// TIA Portal V18 export
VAR_GLOBAL   // PLC tag table "Default tag table_1"
   System_Byte AT %MB1 : Byte;
   FirstScan AT %M1.0 : Bool;
   DiagStatusUpdate AT %M1.1 : Bool;
   AlwaysTRUE AT %M1.2 : Bool;
   AlwaysFALSE AT %M1.3 : Bool;
   Clock_Byte AT %MB0 : Byte;
   Clock_10Hz AT %M0.0 : Bool;
   Clock_5Hz AT %M0.1 : Bool;
   "Clock_2.5Hz" AT %M0.2 : Bool;
   Clock_2Hz AT %M0.3 : Bool;
   "Clock_1.25Hz" AT %M0.4 : Bool;
   Clock_1Hz AT %M0.5 : Bool;
   "Clock_0.625Hz" AT %M0.6 : Bool;
   "Clock_0.5Hz" AT %M0.7 : Bool;
   "H/SSR_019_START" AT %M2.0 : Bool;
   "H/SSR_019_SP" AT %MD4 : Real;
   "H/SSR_019_TT01_PV" AT %MD8 : Real;
   "H/SSR_019_ALERT_SP" AT %MD12 : Real;
   "H/SSR_019_CHBr_RT_SP" AT %MD16 : Real;
   "H/SSR_019_RT_HW_SP" AT %MD20 : Real;
   "H/SSR_019_HW_STEAM_SP" AT %MD24 : Real;
   "H/SSR_019_RT_CHBr_SP" AT %MD28 : Real;
   "H/SSR_019_SOURCE_SEL" AT %MW32 : Int;
   "H/SSR_019_AM" AT %M2.1 : Bool;
   "H/SSR_019_TIME_SP" AT %MW34 : Int;
   "H/SSR_019_KP" AT %MW36 : Int;
   "H/SSR_019_TI" AT %MW38 : Int;
   "H/SSR_019_TT02_PV" AT %MD40 : Real;
   "H/SSR_019_CV02_MANOUT" AT %MD44 : Real;
   "H/SSR_019_START_PV" AT %MD48 : Real;
   "H/SSR_019_CV02_SCVOUT" AT %MD52 : Real;
   "H/SSR_019_RUN_MIN" AT %MW56 : Int;
   "H/SSR_019_FLUSH_TIME_SP" AT %MW60 : Int;
   "H/SSR_019_VENT_TIME_SP" AT %MW62 : Int;
   "H/SSR_019_CONDENSATE_TIME_SP" AT %MW64 : Int;
   "H/SSR_019_XV01_CMD" AT %M58.7 : Bool;
   "H/SSR_019_XV02_CMD" AT %M59.0 : Bool;
   "H/SSR_019_XV03_CMD" AT %M59.1 : Bool;
   "H/SSR_019_XV07_CMD" AT %M59.2 : Bool;
   "H/SSR_019_XV08_CMD" AT %M59.3 : Bool;
   "H/SSR_019_XV09_CMD" AT %M59.4 : Bool;
   "H/SSR_019_XV11_CMD" AT %M59.5 : Bool;
   "H/SSR_019_XV12_CMD" AT %M59.6 : Bool;
   "H/SSR_019_XV13_CMD" AT %M59.7 : Bool;
   "H/SSR_019_XV10_CMD" AT %M66.0 : Bool;
   "H/SSR_019_XV05_CMD" AT %M66.1 : Bool;
   "H/SSR_019_XV06_CMD" AT %M66.2 : Bool;
   "H/SSR_019_FLUSH_RUN_TIME" AT %MD68 : Real;
   "H/SSR_019_CONDENSATE_RUN_TIME" AT %MD72 : Real;
   "H/SSR_019_VENT_RUN_TIME" AT %MD76 : Real;
   "H/SSR_019_CV01_MANOUT" AT %MD80 : Real;
   "H/SSR_019_CV01_SCVOUT" AT %MD84 : Real;
   "H/SSR_019_HOLD" AT %M66.3 : Bool;
   "H/SSR_019_EMSTOP" AT %M66.4 : Bool;
   XV_ERRORMON_TIME AT %MD88 : Time;
   "H/SSR_019_XV01_RESET" AT %M66.5 : Bool;
   "H/SSR_019_XV01_MCMD" AT %M66.6 : Bool;
   "H/SSR_019_XV01_Status" AT %MW92 : Word;
   "H/SSR_019_XV02_MCMD" AT %M66.7 : Bool;
   "H/SSR_019_XV02_RESET" AT %M67.0 : Bool;
   "H/SSR_019_XV03_MCMD" AT %M67.1 : Bool;
   "H/SSR_019_XV03_RESET" AT %M67.2 : Bool;
   "H/SSR_019_XV04_MCMD" AT %M67.3 : Bool;
   "H/SSR_019_XV04_RESET" AT %M67.4 : Bool;
   "H/SSR_019_XV05_MCMD" AT %M67.5 : Bool;
   "H/SSR_019_XV05_RESET" AT %M67.6 : Bool;
   "H/SSR_019_XV06_MCMD" AT %M67.7 : Bool;
   "H/SSR_019_XV06_RESET" AT %M94.0 : Bool;
   "H/SSR_019_XV07_MCMD" AT %M94.1 : Bool;
   "H/SSR_019_XV07_RESET" AT %M94.2 : Bool;
   "H/SSR_019_XV08_MCMD" AT %M94.3 : Bool;
   "H/SSR_019_XV08_RESET" AT %M94.4 : Bool;
   "H/SSR_019_XV09_MCMD" AT %M94.5 : Bool;
   "H/SSR_019_XV09_RESET" AT %M94.6 : Bool;
   "H/SSR_019_XV10_MCMD" AT %M94.7 : Bool;
   "H/SSR_019_XV10_RESET" AT %M95.0 : Bool;
   "H/SSR_019_XV11_MCMD" AT %M95.1 : Bool;
   "H/SSR_019_XV11_RESET" AT %M95.2 : Bool;
   "H/SSR_019_XV12_MCMD" AT %M95.3 : Bool;
   "H/SSR_019_XV12_RESET" AT %M95.4 : Bool;
   "H/SSR_019_XV13_MCMD" AT %M95.5 : Bool;
   "H/SSR_019_XV13_RESET" AT %M95.6 : Bool;
   "H/SSR_019_XV02_Status" AT %MW96 : Word;
   "H/SSR_019_XV03_Status" AT %MW98 : Word;
   "H/SSR_019_XV04_Status" AT %MW100 : Word;
   "H/SSR_019_XV05_Status" AT %MW102 : Word;
   "H/SSR_019_XV07_Status" AT %MW104 : Word;
   "H/SSR_019_XV08_Status" AT %MW106 : Word;
   "H/SSR_019_XV09_Status" AT %MW108 : Word;
   "H/SSR_019_XV10_Status" AT %MW110 : Word;
   "H/SSR_019_XV06_Status" AT %MW112 : Word;
   "H/SSR_019_XV11_Status" AT %MW114 : Word;
   "H/SSR_019_XV12_Status" AT %MW116 : Word;
   "H/SSR_019_XV13_Status" AT %MW118 : Word;
   "H/SSR_019_CV03_SCVOUT" AT %MW120 : Int;
   "H/SSR_019_APT01_PV" AT %MD122 : Real;
   "H/SSR_019_AG_CMD" AT %M2.2 : Bool;
   "H/SSR_019_AG_MCMD" AT %M2.3 : Bool;
   "H/SSR_019_AG_RESET" AT %M2.4 : Bool;
   "H/SSR_019_AG_Status" AT %MW126 : Word;
   "H/SSR_019_CV03_MANOUT" AT %MD128 : Real;
   "H/SSR_019_TT01_Faulty" AT %M2.5 : Bool;
   "H/SSR_019_APT01_Faulty" AT %M2.6 : Bool;
   "H/SSR_019_TT02_Faulty" AT %M2.7 : Bool;
   "H/SSR_019_TT01_Fault" AT %M3.0 : Bool;
   "H/SSR_019_ALERT_SP_EMPTY" AT %M3.1 : Bool;
   "H/SSR_019_SP_EMPTY" AT %M3.2 : Bool;
   "H/SSR_019_CHANGEOVER_SP_EMPTY" AT %M3.3 : Bool;
   "H/SSR_019_FlushTime_SP_EMPTY" AT %M3.4 : Bool;
   "H/SSR_019_VentTime_SP_EMPTY" AT %M3.5 : Bool;
   "H/SSR_019_Cond_Time_EMPTY" AT %M3.6 : Bool;
   "H/SSR_019_XV01_Faulty" AT %M3.7 : Bool;
   "H/SSR_019_XV02_Faulty" AT %M58.0 : Bool;
   "H/SSR_019_XV03_Faulty" AT %M58.1 : Bool;
   "H/SSR_019_XV04_Faulty" AT %M58.2 : Bool;
   "H/SSR_019_XV05_Faulty" AT %M58.3 : Bool;
   "H/SSR_019_XV06_Faulty" AT %M58.4 : Bool;
   "H/SSR_019_XV07_Faulty" AT %M58.5 : Bool;
   "H/SSR_019_XV08_Faulty" AT %M58.6 : Bool;
   "H/SSR_019_XV09_Faulty" AT %M95.7 : Bool;
   "H/SSR_019_XV10_Faulty" AT %M132.0 : Bool;
   "H/SSR_019_XV11_Faulty" AT %M132.1 : Bool;
   "H/SSR_019_XV12_Faulty" AT %M132.2 : Bool;
   "H/SSR_019_XV13_Faulty" AT %M132.3 : Bool;
   "H/SSR_019_Flush_CMP" AT %M132.4 : Bool;
   "H/SSR_019_Vent_CMP" AT %M132.5 : Bool;
   "H/SSR_019_Cond_CMP" AT %M134.0 : Bool;
   "H/SSR_019_GPT101_Fault" AT %M134.1 : Bool;
   "H/SSR_019_GPT101_PV" AT %MD130 : Real;
   "H/SSR_019_GPT201_PV" AT %MD134 : Real;
   "H/SSR_019_GPT201_Fault" AT %M134.2 : Bool;
   "H/SSR_019_GPT301_Fault" AT %M134.3 : Bool;
   "H/SSR_019_GPT401_Fault" AT %M134.4 : Bool;
   "H/SSR_019_GPT501_Fault" AT %M134.5 : Bool;
   "H/SSR_019_GPT601_Fault" AT %M134.6 : Bool;
   "H/SSR_019_TT03_Fault" AT %M135.0 : Bool;
   "H/SSR_019_GPT301_PV" AT %MD132 : Real;
   "H/SSR_019_GPT401_PV" AT %MD135 : Real;
   "H/SSR_019_GPT501_PV" AT %MD136 : Real;
   "H/SSR_019_GPT601_PV" AT %MD137 : Real;
   "H/SSR_019_RESET" AT %M134.7 : Bool;
   "H/SSR_019_TT103_PV" AT %MD138 : Real;
   "H/SSR_019_HOOTER_Status" AT %M135.1 : Bool;
END_VAR
VAR_GLOBAL CONSTANT   // user constants
   "None(1)" : Pip := 65535;
   "Automatic update(1)" : Pip := 0;
   "PIP 1(1)" : Pip := 1;
   "PIP 2(1)" : Pip := 2;
   "PIP 3(1)" : Pip := 3;
   "PIP 4(1)" : Pip := 4;
   "PIP 5(1)" : Pip := 5;
   "PIP 6(1)" : Pip := 6;
   "PIP 7(1)" : Pip := 7;
   "PIP 8(1)" : Pip := 8;
   "PIP 9(1)" : Pip := 9;
   "PIP 10(1)" : Pip := 10;
   "PIP 11(1)" : Pip := 11;
   "PIP 12(1)" : Pip := 12;
   "PIP 13(1)" : Pip := 13;
   "PIP 14(1)" : Pip := 14;
   "PIP 15(1)" : Pip := 15;
   "PIP 16(1)" : Pip := 16;
   "PIP 17(1)" : Pip := 17;
   "PIP 18(1)" : Pip := 18;
   "PIP 19(1)" : Pip := 19;
   "PIP 20(1)" : Pip := 20;
   "PIP 21(1)" : Pip := 21;
   "PIP 22(1)" : Pip := 22;
   "PIP 23(1)" : Pip := 23;
   "PIP 24(1)" : Pip := 24;
   "PIP 25(1)" : Pip := 25;
   "PIP 26(1)" : Pip := 26;
   "PIP 27(1)" : Pip := 27;
   "PIP 28(1)" : Pip := 28;
   "PIP 29(1)" : Pip := 29;
   "PIP 30(1)" : Pip := 30;
   "PIP 31(1)" : Pip := 31;
   "Local1~MC" : Hw_SubModule := 65151;
   "Local1~Common" : Hw_SubModule := 65150;
   "Local1~Device" : Hw_Device := 65132;
   "Local1~Configuration" : Hw_SubModule := 65133;
   "Local1~RHSystem" : Hw_Device := 34;
   "Local1~Display" : Hw_SubModule := 65154;
   "Local1~Exec" : Hw_SubModule := 65152;
   Local1 : Hw_SubModule := 65149;
   "Local1~PROFINET_interface_1" : Hw_Interface := 65164;
   "Local1~PROFINET_interface_1~Port_1" : Hw_Interface := 65165;
   "Local1~PROFINET_interface_1~Port_2" : Hw_Interface := 65166;
   "Local1~PROFINET_interface_1~HsystemIPRef_1" : Hw_Interface := 257;
   "Local1~HCPUredCtrl" : Hw_SubModule := 65147;
   "Local2~MC" : Hw_SubModule := 65351;
   "Local2~Common" : Hw_SubModule := 65350;
   "Local2~Device" : Hw_Device := 65332;
   "Local2~Configuration" : Hw_SubModule := 65333;
   "Local2~Display" : Hw_SubModule := 65354;
   "Local2~Exec" : Hw_SubModule := 65352;
   Local2 : Hw_SubModule := 65349;
   "Local2~PROFINET_interface_1" : Hw_Interface := 65364;
   "Local2~PROFINET_interface_1~Port_1" : Hw_Interface := 65365;
   "Local2~PROFINET_interface_1~Port_2" : Hw_Interface := 65366;
   "Local2~PROFINET_interface_1~HsystemIPRef_1" : Hw_Interface := 268;
   "Local2~HCPUredCtrl" : Hw_SubModule := 65347;
   "OB_AutoLogic(1)" : OB_PCYCLE := 1;
   "OB_Main(1)" : OB_PCYCLE := 123;
   "OB_PID Cyclic interrupt(1)" : OB_Cyclic := 30;
   "OB_Cyclic interrupt(1)" : OB_Cyclic := 31;
END_VAR
